{attribute 'linkalways'} 
{attribute 'no_explicit_call' := 'This FB is a CLASS and must be accessed using methods or properties'}
{attribute 'enable_dynamic_creation'}
FUNCTION_BLOCK SetPositionCommand EXTENDS Mc2AxisCommand
VAR
	_position : LREAL;
	_mode : SetPositionMode;
END_VAR

METHOD FB_init : BOOL
VAR_INPUT
	bInitRetains : BOOL; // if TRUE, the retain variables are initialized (warm start / cold start)
	bInCopyCode : BOOL;  // if TRUE, the instance afterwards gets moved into the copy code (online change)
	axis : Axis;
	position : LREAL;
	mode : SetPositionMode;
END_VAR
_axis := axis;
_position := position;
_mode := mode;
END_METHOD

METHOD PROTECTED OnExecuting
VAR_INPUT
	stateControl : I_AsyncCommandStateControl;
END_VAR
VAR_INST
	_fb : MC_SetPosition;
END_VAR
_fb(
	Axis := _axis._InternalAxisRef,
	Execute := TRUE,
	Position := _position,
	Mode := (_mode = SetPositionMode.Relative)
);

IF _fb.Busy THEN
	RETURN;
END_IF

_fb(Axis := _axis._InternalAxisRef, Execute := FALSE);

IF _fb.Error THEN
	stateControl.Error(_fb.ErrorID);
	RETURN;
END_IF

stateControl.Next();
END_METHOD

END_FUNCTION_BLOCK

(* stored: Version 1.1.0.1, ProductVersion 3.1.4026.13
   POU SetPositionCommand: Id {2a902d1c-fb1d-03bf-185a-32f82cc2898f}, SpecialFunc None
   Folder Constructor: Id {6f4dfddd-479c-0ff2-0b84-3cb3374b4990}
   Method FB_init: Id {982f49f2-3964-0581-0af5-dc2bc19317cf}
   Method OnExecuting: Id {f5066999-4a47-0b87-3ed1-c4cb4e3ffff9} *)
